FUNCTION_BLOCK OF_E_TABLE (* Composite Function Block Type *)
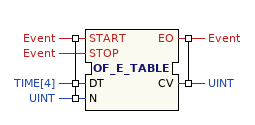
  EVENT_INPUT
    START WITH DT, N; (* Start table driven event generation *)
    STOP; (* Stop table driven event generation *)
  END_EVENT
  EVENT_OUTPUT
    EO WITH CV; (* Generated events: N events at periods DT, starting at DT[0] after START *)
  END_EVENT
  VAR_INPUT
    DT : ARRAY [0..3] OF TIME; (* Periods between events *)
    N : UINT; (* Number of events to generate *)
  END_VAR
  VAR_OUTPUT
    CV : UINT; (* Current event index, 0..N-1 *)
  END_VAR
END_FUNCTION_BLOCK
